Yaskawa INFORM job: pipe_uncentered_cylinder_program.JBI

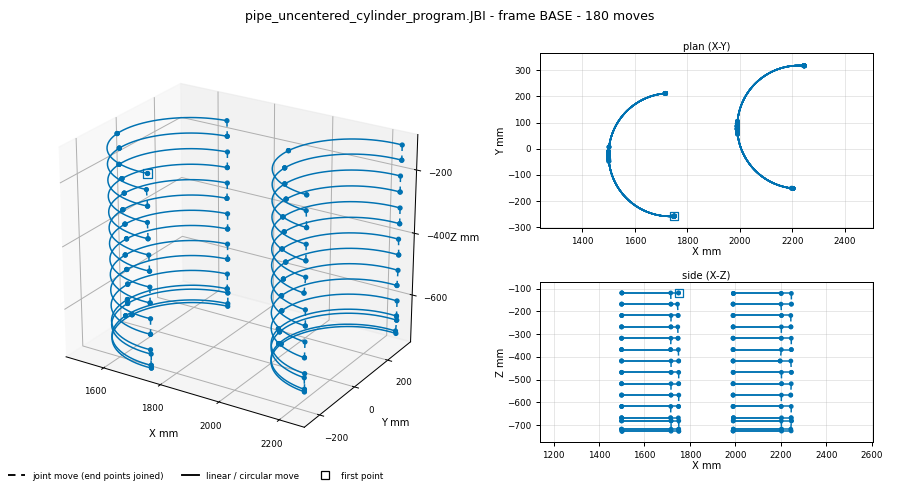
[picture p0: tool path of pipe_uncentered_cylinder_program.JBI in frame BASE, 180 of 245 moves have a stored position in this frame; points joined in program order, loops and branches not executed]
/JOB
//NAME pipe_uncentered_cylinder_program
//POS
///NPOS 240,0,240,0,0,0
///TOOL 0
///POSTYPE BASE
///RECTAN
///RCONF 0,0,0,0,0,0,0,0,0,0,0,0,0,0,0,0,0,0,0,0,0,0,0,0
C00000=1749.940904,-257.239351,-118.539050,-86.127714,-90.000000,5.000000
C00001=1749.940904,-257.239351,-118.539050,-86.127714,-90.000000,5.000000
C00002=1591.453481,-209.463262,-118.539050,-127.423189,-89.999999,5.000000
C00003=1500.680855,-47.796008,-118.539050,-173.950296,-90.000000,5.000000
C00004=1500.680855,-47.796008,-118.539050,-173.950296,-90.000000,5.000000
C00005=1500.680855,-47.796008,-118.539050,-173.950296,-90.000000,5.000000
C00006=1545.974830,117.313444,-118.539050,143.269507,-90.000000,5.000000
C00007=1715.536670,210.922784,-118.539050,94.533692,-90.000000,5.000000
C00008=1716.466846,210.994681,-167.787500,94.305952,-89.999999,5.000000
C00009=1716.466846,210.994681,-167.787500,94.305952,-89.999999,5.000000
C00010=1554.324971,127.859099,-167.787500,139.985523,-89.999999,5.000000
C00011=1499.816295,-37.466638,-167.787500,-175.000000,-90.000000,5.000000
C00012=1499.816295,-37.466638,-167.787500,-175.000000,-90.000000,5.000000
C00013=1499.816295,-37.466638,-167.787500,-175.000000,-90.000000,5.000000
C00014=1575.986813,-196.538427,-167.787500,-132.344944,-90.000000,5.000000
C00015=1745.242286,-257.510095,-167.787500,-87.276599,-90.000000,5.000000
C00016=1747.956735,-257.365215,-217.741000,-86.613037,-90.000000,5.000000
C00017=1747.956735,-257.365215,-217.741000,-86.613037,-90.000000,5.000000
C00018=1577.099305,-197.545821,-217.741000,-131.978582,-89.999999,5.000000
C00019=1500.085421,-41.323879,-217.741000,-175.000000,-89.999999,5.000000
C00020=1500.085421,-41.323879,-217.741000,-175.000000,-89.999999,5.000000
C00021=1500.085421,-41.323879,-217.741000,-175.000000,-89.999999,5.000000
C00022=1562.652474,137.256037,-217.741000,136.920187,-90.000000,5.000000
C00023=1717.040812,211.037190,-217.741000,94.165460,-90.000000,5.000000
C00024=1716.357109,210.986393,-267.822500,94.332816,-90.000000,5.000000
C00025=1716.357109,210.986393,-267.822500,94.332816,-90.000000,5.000000
C00026=1562.860730,137.478452,-267.822500,136.845809,-90.000000,5.000000
C00027=1499.417640,-27.601325,-267.822500,-175.000000,-90.000000,5.000000
C00028=1499.417640,-27.601325,-267.822500,-175.000000,-90.000000,5.000000
C00029=1499.417640,-27.601325,-267.822500,-175.000000,-90.000000,5.000000
C00030=1572.172718,-192.984054,-267.822500,-133.617628,-90.000000,5.000000
C00031=1746.492309,-257.447293,-267.822500,-86.971075,-90.000000,5.000000
C00032=1747.500808,-257.391753,-317.748500,-86.724521,-90.000000,5.000000
C00033=1747.500808,-257.391753,-317.748500,-86.724521,-90.000000,5.000000
C00034=1571.275066,-192.124158,-317.748500,-133.921067,-89.999999,5.000000
C00035=1499.445999,-17.233020,-317.748500,175.000000,-90.000000,5.000000
C00036=1499.445999,-17.233020,-317.748500,175.000000,-90.000000,5.000000
C00037=1499.445999,-17.233020,-317.748500,175.000000,-90.000000,5.000000
C00038=1566.953470,141.735162,-317.748500,135.404299,-90.000000,5.000000
C00039=1716.359373,210.986564,-317.748500,94.332262,-90.000000,5.000000
C00040=1715.055844,210.884161,-367.795500,94.651443,-90.000000,5.000000
C00041=1715.055844,210.884161,-367.795500,94.651443,-90.000000,5.000000
C00042=1568.265848,143.055676,-367.795500,134.949834,-89.999999,5.000000
C00043=1499.396571,-26.336761,-367.795500,-175.000000,-89.999999,5.000000
C00044=1499.396571,-26.336761,-367.795500,-175.000000,-89.999999,5.000000
C00045=1499.396571,-26.336761,-367.795500,-175.000000,-89.999999,5.000000
C00046=1569.975341,-190.862783,-367.795500,-134.363188,-90.000000,5.000000
C00047=1748.987493,-257.301936,-367.795500,-86.360949,-90.000000,5.000000
C00048=1750.526532,-257.198976,-417.775000,-85.984419,-90.000000,5.000000
C00049=1750.526532,-257.198976,-417.775000,-85.984419,-90.000000,5.000000
C00050=1569.600086,-190.494955,-417.775000,-134.491458,-90.000000,5.000000
C00051=1499.446271,-17.222088,-417.775000,175.000000,-90.000000,5.000000
C00052=1499.446271,-17.222088,-417.775000,175.000000,-90.000000,5.000000
C00053=1499.446271,-17.222088,-417.775000,175.000000,-90.000000,5.000000
C00054=1570.664090,145.415647,-417.775000,134.128488,-90.000000,5.000000
C00055=1716.962407,211.031467,-417.775000,94.184650,-90.000000,5.000000
C00056=1717.005411,211.034610,-467.823500,94.174124,-90.000000,5.000000
C00057=1717.005411,211.034610,-467.823500,94.174124,-90.000000,5.000000
C00058=1563.073398,137.704983,-467.823500,136.769961,-89.999999,5.000000
C00059=1499.674917,-11.171269,-467.823500,175.000000,-90.000000,5.000000
C00060=1499.674917,-11.171269,-467.823500,175.000000,-90.000000,5.000000
C00061=1499.674917,-11.171269,-467.823500,175.000000,-90.000000,5.000000
C00062=1571.299255,-192.147450,-467.823500,-133.912870,-90.000000,5.000000
C00063=1750.593496,-257.194266,-467.823500,-85.968032,-90.000000,5.000000
C00064=1750.562997,-257.196413,-517.742500,-85.975495,-90.000000,5.000000
C00065=1750.562997,-257.196413,-517.742500,-85.975495,-90.000000,5.000000
C00066=1569.533050,-190.429072,-517.742500,-134.514402,-90.000000,5.000000
C00067=1499.402780,-19.363326,-517.742500,175.000000,-89.999999,5.000000
C00068=1499.402780,-19.363326,-517.742500,175.000000,-89.999999,5.000000
C00069=1499.402780,-19.363326,-517.742500,175.000000,-89.999999,5.000000
C00070=1567.369334,142.155874,-517.742500,135.259896,-89.999999,5.000000
C00071=1716.613272,211.005660,-517.742500,94.270109,-89.999999,5.000000
C00072=1716.823581,211.021268,-567.815000,94.218629,-90.000000,5.000000
C00073=1716.823581,211.021268,-567.815000,94.218629,-90.000000,5.000000
C00074=1567.685117,142.473927,-567.815000,135.150489,-90.000000,5.000000
C00075=1499.562947,-13.635054,-567.815000,175.000000,-89.999999,5.000000
C00076=1499.562947,-13.635054,-567.815000,175.000000,-89.999999,5.000000
C00077=1499.562947,-13.635054,-567.815000,175.000000,-89.999999,5.000000
C00078=1560.121142,-180.623494,-567.815000,-137.832681,-90.000000,5.000000
C00079=1751.024331,-257.163499,-567.815000,-85.862594,-90.000000,5.000000
C00080=1750.015796,-257.234270,-617.780500,-86.109390,-89.999999,5.000000
C00081=1750.015796,-257.234270,-617.780500,-86.109390,-89.999999,5.000000
C00082=1559.512787,-179.949185,-617.780500,-138.054373,-90.000000,5.000000
C00083=1499.705471,-10.583354,-617.780500,175.000000,-90.000000,5.000000
C00084=1499.705471,-10.583354,-617.780500,175.000000,-90.000000,5.000000
C00085=1499.705471,-10.583354,-617.780500,175.000000,-90.000000,5.000000
C00086=1570.812903,145.559872,-617.780500,134.077900,-90.000000,5.000000
C00087=1715.782793,210.942170,-617.780500,94.473426,-89.999999,5.000000
C00088=1715.115153,210.888979,-667.838500,94.636917,-90.000000,5.000000
C00089=1715.115153,210.888979,-667.838500,94.636917,-90.000000,5.000000
C00090=1572.298871,146.986185,-667.838500,133.575106,-90.000000,5.000000
C00091=1499.565682,-13.567229,-667.838500,175.000000,-90.000000,5.000000
C00092=1499.565682,-13.567229,-667.838500,175.000000,-90.000000,5.000000
C00093=1499.565682,-13.567229,-667.838500,175.000000,-90.000000,5.000000
C00094=1567.110596,-188.012358,-667.838500,-135.349696,-90.000000,5.000000
C00095=1749.049055,-257.298013,-667.838500,-86.345891,-90.000000,5.000000
C00096=1750.503472,-257.200594,-717.761000,-85.990062,-90.000000,5.000000
C00097=1750.503472,-257.200594,-717.761000,-85.990062,-90.000000,5.000000
C00098=1567.704779,-188.611679,-717.761000,-135.143684,-90.000000,5.000000
C00099=1499.381472,-24.971037,-717.761000,-175.000000,-90.000000,5.000000
C00100=1499.381472,-24.971037,-717.761000,-175.000000,-90.000000,5.000000
C00101=1499.381472,-24.971037,-717.761000,-175.000000,-90.000000,5.000000
C00102=1562.233334,136.806640,-717.761000,137.070196,-90.000000,5.000000
C00103=1717.054447,211.038183,-717.761000,94.162123,-89.999999,5.000000
C00104=1717.121726,211.043069,-681.141960,-175.000000,-60.000000,-85.854344
C00105=1717.121726,211.043069,-681.141960,-175.000000,-60.000000,-85.854344
C00106=1567.606056,142.394412,-681.141960,-175.000000,-60.000000,-44.822139
C00107=1499.579001,-13.243673,-681.141960,175.000000,-60.000000,-5.000000
C00108=1499.579001,-13.243673,-681.141960,175.000000,-60.000000,-5.000000
C00109=1499.579001,-13.243673,-681.141960,175.000000,-60.000000,-5.000000
C00110=1566.014614,-186.895493,-681.141960,175.000000,-60.000000,44.268328
C00111=1750.849014,-257.176115,-681.141960,175.000000,-60.000000,94.094499
C00112=1751.015595,-257.164131,-726.640960,175.000000,-60.000000,94.135268
C00113=1751.015595,-257.164131,-726.640960,175.000000,-60.000000,94.135268
C00114=1552.700260,-172.020396,-726.640960,-175.000000,-60.000000,39.393640
C00115=1501.257028,6.615173,-726.640960,175.000000,-60.000000,-7.263097
C00116=1501.257028,6.615173,-726.640960,175.000000,-60.000000,-7.263097
C00117=1501.257028,6.615173,-726.640960,175.000000,-60.000000,-7.263097
C00118=1579.136007,153.239023,-726.640960,175.000000,-60.000000,-48.686744
C00119=1716.838691,211.022382,-726.640960,-175.000000,-60.000000,-85.785069
C00120=2201.495182,-151.068736,-120.674700,-95.658348,-90.000000,5.000000
C00121=2201.495182,-151.068736,-120.674700,-95.658348,-90.000000,5.000000
C00122=2044.257197,-67.678403,-120.674700,-140.219665,-90.000000,5.000000
C00123=1990.979209,104.765230,-120.674700,174.557660,-90.000000,5.000000
C00124=1990.979209,104.765230,-120.674700,174.557660,-90.000000,5.000000
C00125=1990.979209,104.765230,-120.674700,174.557660,-90.000000,5.000000
C00126=2064.299554,253.919936,-120.674700,133.087419,-90.000000,5.000000
C00127=2246.112616,316.235511,-120.674700,84.750402,-90.000000,5.000000
C00128=2246.169004,316.230323,-167.736500,84.736579,-90.000000,5.000000
C00129=2246.169004,316.230323,-167.736500,84.736579,-90.000000,5.000000
C00130=2063.146664,252.834241,-167.736500,133.473995,-90.000000,5.000000
C00131=1989.947901,86.047865,-167.736500,175.000000,-89.999999,5.000000
C00132=1989.947901,86.047865,-167.736500,175.000000,-89.999999,5.000000
C00133=1989.947901,86.047865,-167.736500,175.000000,-89.999999,5.000000
C00134=2052.059148,-76.582521,-167.736500,-137.329465,-89.999999,5.000000
C00135=2200.564996,-150.974703,-167.736500,-95.886570,-90.000000,5.000000
C00136=2202.695265,-151.184528,-217.738500,-95.364039,-89.999999,5.000000
C00137=2202.695265,-151.184528,-217.738500,-95.364039,-89.999999,5.000000
C00138=2049.346534,-73.588554,-217.738500,-138.315683,-90.000000,5.000000
C00139=1989.967085,87.147586,-217.738500,175.000000,-90.000000,5.000000
C00140=1989.967085,87.147586,-217.738500,175.000000,-90.000000,5.000000
C00141=1989.967085,87.147586,-217.738500,175.000000,-90.000000,5.000000
C00142=2060.819888,250.597642,-217.738500,134.261837,-89.999999,5.000000
C00143=2243.608192,316.452099,-217.738500,85.364033,-90.000000,5.000000
C00144=2244.039674,316.416710,-267.790000,85.258352,-90.000000,5.000000
C00145=2244.039674,316.416710,-267.790000,85.258352,-90.000000,5.000000
C00146=2071.779846,260.622536,-267.790000,130.635454,-89.999999,5.000000
C00147=1990.257189,95.059201,-267.790000,175.000000,-89.999999,5.000000
C00148=1990.257189,95.059201,-267.790000,175.000000,-89.999999,5.000000
C00149=1990.257189,95.059201,-267.790000,175.000000,-89.999999,5.000000
C00150=2049.513988,-73.776402,-267.790000,-138.254254,-90.000000,5.000000
C00151=2202.070096,-151.124984,-267.790000,-95.517338,-89.999999,5.000000
C00152=2201.732367,-151.092115,-317.761500,-95.600169,-90.000000,5.000000
C00153=2201.732367,-151.092115,-317.761500,-95.600169,-90.000000,5.000000
C00154=2058.339900,-83.136929,-317.761500,-135.113353,-90.000000,5.000000
C00155=1989.951054,78.756762,-317.761500,-175.000000,-90.000000,5.000000
C00156=1989.951054,78.756762,-317.761500,-175.000000,-90.000000,5.000000
C00157=1989.951054,78.756762,-317.761500,-175.000000,-90.000000,5.000000
C00158=2070.732503,259.718356,-317.761500,130.973211,-90.000000,5.000000
C00159=2245.637578,316.278670,-317.761500,84.866839,-90.000000,5.000000
C00160=2246.012474,316.244690,-367.767000,84.774950,-89.999999,5.000000
C00161=2246.012474,316.244690,-367.767000,84.774950,-89.999999,5.000000
C00162=2061.479430,251.237892,-367.767000,134.037456,-89.999999,5.000000
C00163=1989.955586,86.524700,-367.767000,175.000000,-90.000000,5.000000
C00164=1989.955586,86.524700,-367.767000,175.000000,-90.000000,5.000000
C00165=1989.955586,86.524700,-367.767000,175.000000,-90.000000,5.000000
C00166=2045.484077,-69.139856,-367.767000,-139.753869,-89.999999,5.000000
C00167=2201.922845,-151.110713,-367.767000,-95.553451,-90.000000,5.000000
C00168=2196.726495,-150.546997,-417.788500,-96.829383,-90.000000,5.000000
C00169=2196.726495,-150.546997,-417.788500,-96.829383,-90.000000,5.000000
C00170=2053.431275,-78.058253,-417.788500,-136.837571,-90.000000,5.000000
C00171=1990.036838,75.135124,-417.788500,-175.000000,-89.999999,5.000000
C00172=1990.036838,75.135124,-417.788500,-175.000000,-89.999999,5.000000
C00173=1990.036838,75.135124,-417.788500,-175.000000,-89.999999,5.000000
C00174=2058.402661,248.207538,-417.788500,135.091648,-90.000000,5.000000
C00175=2243.881899,316.429743,-417.788500,85.296997,-89.999999,5.000000
C00176=2246.061371,316.240213,-467.763000,84.762964,-90.000000,5.000000
C00177=2246.061371,316.240213,-467.763000,84.762964,-90.000000,5.000000
C00178=2071.679385,260.536273,-467.763000,130.667777,-90.000000,5.000000
C00179=1990.326877,96.298740,-467.763000,175.000000,-90.000000,5.000000
C00180=1990.326877,96.298740,-467.763000,175.000000,-90.000000,5.000000
C00181=1990.326877,96.298740,-467.763000,175.000000,-90.000000,5.000000
C00182=2052.360794,-76.909127,-467.763000,-137.220937,-90.000000,5.000000
C00183=2202.313125,-151.148331,-467.763000,-95.457740,-90.000000,5.000000
C00184=2202.902488,-151.203892,-517.762500,-95.313234,-90.000000,5.000000
C00185=2202.902488,-151.203892,-517.762500,-95.313234,-90.000000,5.000000
C00186=2057.105877,-81.888713,-517.762500,-135.541819,-89.999999,5.000000
C00187=1989.931219,84.678581,-517.762500,175.000000,-89.999999,5.000000
C00188=1989.931219,84.678581,-517.762500,175.000000,-89.999999,5.000000
C00189=1989.931219,84.678581,-517.762500,175.000000,-89.999999,5.000000
C00190=2068.385658,257.652621,-517.762500,131.736413,-89.999999,5.000000
C00191=2245.482409,316.292557,-517.762500,84.904869,-90.000000,5.000000
C00192=2243.362690,316.471877,-567.772500,85.424156,-90.000000,5.000000
C00193=2243.362690,316.471877,-567.772500,85.424156,-90.000000,5.000000
C00194=2051.378042,240.848086,-567.772500,137.575342,-90.000000,5.000000
C00195=1990.060890,74.405537,-567.772500,-175.000000,-89.999999,5.000000
C00196=1990.060890,74.405537,-567.772500,-175.000000,-89.999999,5.000000
C00197=1990.060890,74.405537,-567.772500,-175.000000,-89.999999,5.000000
C00198=2061.322668,-86.078546,-567.772500,-134.090710,-89.999999,5.000000
C00199=2202.327386,-151.149694,-567.772500,-95.454242,-90.000000,5.000000
C00200=2201.367177,-151.056018,-617.754500,-95.689749,-90.000000,5.000000
C00201=2201.367177,-151.056018,-617.754500,-95.689749,-90.000000,5.000000
C00202=2052.658725,-77.230498,-617.754500,-137.113963,-90.000000,5.000000
C00203=1989.999951,76.421959,-617.754500,-175.000000,-89.999999,5.000000
C00204=1989.999951,76.421959,-617.754500,-175.000000,-89.999999,5.000000
C00205=1989.999951,76.421959,-617.754500,-175.000000,-89.999999,5.000000
C00206=2056.480347,246.256427,-617.754500,135.760260,-90.000000,5.000000
C00207=2245.513226,316.289808,-617.754500,84.897316,-90.000000,5.000000
C00208=2245.267041,316.311660,-667.687000,84.957648,-90.000000,5.000000
C00209=2245.267041,316.311660,-667.687000,84.957648,-90.000000,5.000000
C00210=2046.291839,235.096654,-667.687000,139.449624,-90.000000,5.000000
C00211=1991.451727,55.742592,-667.687000,-173.453172,-89.999999,5.000000
C00212=1991.451727,55.742592,-667.687000,-173.453172,-89.999999,5.000000
C00213=1991.451727,55.742592,-667.687000,-173.453172,-89.999999,5.000000
C00214=2061.762417,-86.503446,-667.687000,-133.941441,-90.000000,5.000000
C00215=2202.791447,-151.193539,-667.687000,-95.340457,-90.000000,5.000000
C00216=2202.766975,-151.191250,-717.769500,-95.346457,-89.999999,5.000000
C00217=2202.766975,-151.191250,-717.769500,-95.346457,-89.999999,5.000000
C00218=2056.491256,-81.260006,-717.769500,-135.756443,-90.000000,5.000000
C00219=1991.056336,59.447196,-717.769500,-174.362636,-89.999999,5.000000
C00220=1991.056336,59.447196,-717.769500,-174.362636,-89.999999,5.000000
C00221=1991.056336,59.447196,-717.769500,-174.362636,-89.999999,5.000000
C00222=2050.583896,239.974736,-717.769500,137.863492,-90.000000,5.000000
C00223=2243.561805,316.455856,-717.769500,85.375394,-89.999999,5.000000
C00224=2246.301849,316.218047,-681.093960,175.000000,-60.000000,-95.295987
C00225=2246.301849,316.218047,-681.093960,175.000000,-60.000000,-95.295987
C00226=2049.280658,238.522168,-681.093960,-175.000000,-60.000000,-41.660131
C00227=1990.652766,63.985921,-681.093960,175.000000,-60.000000,5.000000
C00228=1990.652766,63.985921,-681.093960,175.000000,-60.000000,5.000000
C00229=1990.652766,63.985921,-681.093960,175.000000,-60.000000,5.000000
C00230=2060.887500,-85.655884,-681.093960,175.000000,-60.000000,45.761205
C00231=2201.648298,-151.083856,-681.093960,175.000000,-60.000000,84.379210
C00232=2202.847007,-151.198726,-725.482960,-175.000000,-60.000000,84.673164
C00233=2202.847007,-151.198726,-725.482960,-175.000000,-60.000000,84.673164
C00234=2065.711002,-90.221730,-725.482960,-175.000000,-60.000000,47.382559
C00235=1990.062143,74.369326,-725.482960,175.000000,-60.000000,5.000000
C00236=1990.062143,74.369326,-725.482960,175.000000,-60.000000,5.000000
C00237=1990.062143,74.369326,-725.482960,175.000000,-60.000000,5.000000
C00238=2051.419035,240.892928,-725.482960,175.000000,-60.000000,-42.439489
C00239=2245.154859,316.321531,-725.482960,175.000000,-60.000000,-95.014862
///POSTYPE PULSE
///PULSE
EX00000=80896.0
EX00001=256000.0
///POSTYPE PULSE
///PULSE
EC00000=80896.0
EC00001=80896.0
EC00002=80896.0
EC00003=80896.0
EC00004=80896.0
EC00005=80896.0
EC00006=80896.0
EC00007=80896.0
EC00008=80896.0
EC00009=80896.0
EC00010=80896.0
EC00011=80896.0
EC00012=80896.0
EC00013=80896.0
EC00014=80896.0
EC00015=80896.0
EC00016=80896.0
EC00017=80896.0
EC00018=80896.0
EC00019=80896.0
EC00020=80896.0
EC00021=80896.0
EC00022=80896.0
EC00023=80896.0
EC00024=80896.0
EC00025=80896.0
EC00026=80896.0
EC00027=80896.0
EC00028=80896.0
EC00029=80896.0
EC00030=80896.0
EC00031=80896.0
EC00032=80896.0
EC00033=80896.0
EC00034=80896.0
EC00035=80896.0
EC00036=80896.0
EC00037=80896.0
EC00038=80896.0
EC00039=80896.0
EC00040=80896.0
EC00041=80896.0
EC00042=80896.0
EC00043=80896.0
EC00044=80896.0
EC00045=80896.0
EC00046=80896.0
EC00047=80896.0
EC00048=80896.0
EC00049=80896.0
EC00050=80896.0
EC00051=80896.0
EC00052=80896.0
EC00053=80896.0
EC00054=80896.0
EC00055=80896.0
EC00056=80896.0
EC00057=80896.0
EC00058=80896.0
EC00059=80896.0
EC00060=80896.0
EC00061=80896.0
EC00062=80896.0
EC00063=80896.0
EC00064=80896.0
EC00065=80896.0
EC00066=80896.0
EC00067=80896.0
EC00068=80896.0
EC00069=80896.0
EC00070=80896.0
EC00071=80896.0
EC00072=80896.0
EC00073=80896.0
EC00074=80896.0
EC00075=80896.0
EC00076=80896.0
EC00077=80896.0
EC00078=80896.0
EC00079=80896.0
EC00080=80896.0
EC00081=80896.0
EC00082=80896.0
EC00083=80896.0
EC00084=80896.0
EC00085=80896.0
EC00086=80896.0
EC00087=80896.0
EC00088=80896.0
EC00089=80896.0
EC00090=80896.0
EC00091=80896.0
EC00092=80896.0
EC00093=80896.0
EC00094=80896.0
EC00095=80896.0
EC00096=80896.0
EC00097=80896.0
EC00098=80896.0
EC00099=80896.0
EC00100=80896.0
EC00101=80896.0
EC00102=80896.0
EC00103=80896.0
EC00104=80896.0
EC00105=80896.0
EC00106=80896.0
EC00107=80896.0
EC00108=80896.0
EC00109=80896.0
EC00110=80896.0
EC00111=80896.0
EC00112=80896.0
EC00113=80896.0
EC00114=80896.0
EC00115=80896.0
EC00116=80896.0
EC00117=80896.0
EC00118=80896.0
EC00119=80896.0
EC00120=256000.0
EC00121=256000.0
EC00122=256000.0
EC00123=256000.0
EC00124=256000.0
EC00125=256000.0
EC00126=256000.0
EC00127=256000.0
EC00128=256000.0
EC00129=256000.0
EC00130=256000.0
EC00131=256000.0
EC00132=256000.0
EC00133=256000.0
EC00134=256000.0
EC00135=256000.0
EC00136=256000.0
EC00137=256000.0
EC00138=256000.0
EC00139=256000.0
EC00140=256000.0
EC00141=256000.0
EC00142=256000.0
EC00143=256000.0
EC00144=256000.0
EC00145=256000.0
EC00146=256000.0
EC00147=256000.0
EC00148=256000.0
EC00149=256000.0
EC00150=256000.0
EC00151=256000.0
EC00152=256000.0
EC00153=256000.0
EC00154=256000.0
EC00155=256000.0
EC00156=256000.0
EC00157=256000.0
EC00158=256000.0
EC00159=256000.0
EC00160=256000.0
EC00161=256000.0
EC00162=256000.0
EC00163=256000.0
EC00164=256000.0
EC00165=256000.0
EC00166=256000.0
EC00167=256000.0
EC00168=256000.0
EC00169=256000.0
EC00170=256000.0
EC00171=256000.0
EC00172=256000.0
EC00173=256000.0
EC00174=256000.0
EC00175=256000.0
EC00176=256000.0
EC00177=256000.0
EC00178=256000.0
EC00179=256000.0
EC00180=256000.0
EC00181=256000.0
EC00182=256000.0
EC00183=256000.0
EC00184=256000.0
EC00185=256000.0
EC00186=256000.0
EC00187=256000.0
EC00188=256000.0
EC00189=256000.0
EC00190=256000.0
EC00191=256000.0
EC00192=256000.0
EC00193=256000.0
EC00194=256000.0
EC00195=256000.0
EC00196=256000.0
EC00197=256000.0
EC00198=256000.0
EC00199=256000.0
EC00200=256000.0
EC00201=256000.0
EC00202=256000.0
EC00203=256000.0
EC00204=256000.0
EC00205=256000.0
EC00206=256000.0
EC00207=256000.0
EC00208=256000.0
EC00209=256000.0
EC00210=256000.0
EC00211=256000.0
EC00212=256000.0
EC00213=256000.0
EC00214=256000.0
EC00215=256000.0
EC00216=256000.0
EC00217=256000.0
EC00218=256000.0
EC00219=256000.0
EC00220=256000.0
EC00221=256000.0
EC00222=256000.0
EC00223=256000.0
EC00224=256000.0
EC00225=256000.0
EC00226=256000.0
EC00227=256000.0
EC00228=256000.0
EC00229=256000.0
EC00230=256000.0
EC00231=256000.0
EC00232=256000.0
EC00233=256000.0
EC00234=256000.0
EC00235=256000.0
EC00236=256000.0
EC00237=256000.0
EC00238=256000.0
EC00239=256000.0
//INST
///DATE 2023/08/15 14:21
///ATTR SC,RW,RJ
////FRAME BASE
///GROUP1 RB1,ST1
NOP
MOVJ P009 EX000 VJ=15.00
MOVJ C00000 EC00000 VJ=15.0
CALL JOB:SPYON
MOVC C00001 EC00001 V=150.0
MOVC C00002 EC00002 V=150.0
MOVC C00003 EC00003 V=150.0
MOVJ C00004 EC00004 VJ=15.0
MOVC C00005 EC00005 V=150.0
MOVC C00006 EC00006 V=150.0
MOVC C00007 EC00007 V=150.0
MOVJ C00008 EC00008 VJ=15.0
MOVC C00009 EC00009 V=150.0
MOVC C00010 EC00010 V=150.0
MOVC C00011 EC00011 V=150.0
MOVJ C00012 EC00012 VJ=15.0
MOVC C00013 EC00013 V=150.0
MOVC C00014 EC00014 V=150.0
MOVC C00015 EC00015 V=150.0
MOVJ C00016 EC00016 VJ=15.0
MOVC C00017 EC00017 V=150.0
MOVC C00018 EC00018 V=150.0
MOVC C00019 EC00019 V=150.0
MOVJ C00020 EC00020 VJ=15.0
MOVC C00021 EC00021 V=150.0
MOVC C00022 EC00022 V=150.0
MOVC C00023 EC00023 V=150.0
MOVJ C00024 EC00024 VJ=15.0
MOVC C00025 EC00025 V=150.0
MOVC C00026 EC00026 V=150.0
MOVC C00027 EC00027 V=150.0
MOVJ C00028 EC00028 VJ=15.0
MOVC C00029 EC00029 V=150.0
MOVC C00030 EC00030 V=150.0
MOVC C00031 EC00031 V=150.0
MOVJ C00032 EC00032 VJ=15.0
MOVC C00033 EC00033 V=150.0
MOVC C00034 EC00034 V=150.0
MOVC C00035 EC00035 V=150.0
MOVJ C00036 EC00036 VJ=15.0
MOVC C00037 EC00037 V=150.0
MOVC C00038 EC00038 V=150.0
MOVC C00039 EC00039 V=150.0
MOVJ C00040 EC00040 VJ=15.0
MOVC C00041 EC00041 V=150.0
MOVC C00042 EC00042 V=150.0
MOVC C00043 EC00043 V=150.0
MOVJ C00044 EC00044 VJ=15.0
MOVC C00045 EC00045 V=150.0
MOVC C00046 EC00046 V=150.0
MOVC C00047 EC00047 V=150.0
MOVJ C00048 EC00048 VJ=15.0
MOVC C00049 EC00049 V=150.0
MOVC C00050 EC00050 V=150.0
MOVC C00051 EC00051 V=150.0
MOVJ C00052 EC00052 VJ=15.0
MOVC C00053 EC00053 V=150.0
MOVC C00054 EC00054 V=150.0
MOVC C00055 EC00055 V=150.0
MOVJ C00056 EC00056 VJ=15.0
MOVC C00057 EC00057 V=150.0
MOVC C00058 EC00058 V=150.0
MOVC C00059 EC00059 V=150.0
MOVJ C00060 EC00060 VJ=15.0
MOVC C00061 EC00061 V=150.0
MOVC C00062 EC00062 V=150.0
MOVC C00063 EC00063 V=150.0
MOVJ C00064 EC00064 VJ=15.0
MOVC C00065 EC00065 V=150.0
MOVC C00066 EC00066 V=150.0
MOVC C00067 EC00067 V=150.0
MOVJ C00068 EC00068 VJ=15.0
MOVC C00069 EC00069 V=150.0
MOVC C00070 EC00070 V=150.0
MOVC C00071 EC00071 V=150.0
MOVJ C00072 EC00072 VJ=15.0
MOVC C00073 EC00073 V=150.0
MOVC C00074 EC00074 V=150.0
MOVC C00075 EC00075 V=150.0
MOVJ C00076 EC00076 VJ=15.0
MOVC C00077 EC00077 V=150.0
MOVC C00078 EC00078 V=150.0
MOVC C00079 EC00079 V=150.0
MOVJ C00080 EC00080 VJ=15.0
MOVC C00081 EC00081 V=150.0
MOVC C00082 EC00082 V=150.0
MOVC C00083 EC00083 V=150.0
MOVJ C00084 EC00084 VJ=15.0
MOVC C00085 EC00085 V=150.0
MOVC C00086 EC00086 V=150.0
MOVC C00087 EC00087 V=150.0
MOVJ C00088 EC00088 VJ=15.0
MOVC C00089 EC00089 V=150.0
MOVC C00090 EC00090 V=150.0
MOVC C00091 EC00091 V=150.0
MOVJ C00092 EC00092 VJ=15.0
MOVC C00093 EC00093 V=150.0
MOVC C00094 EC00094 V=150.0
MOVC C00095 EC00095 V=150.0
MOVJ C00096 EC00096 VJ=15.0
MOVC C00097 EC00097 V=150.0
MOVC C00098 EC00098 V=150.0
MOVC C00099 EC00099 V=150.0
MOVJ C00100 EC00100 VJ=15.0
MOVC C00101 EC00101 V=150.0
MOVC C00102 EC00102 V=150.0
MOVC C00103 EC00103 V=150.0
MOVJ C00104 EC00104 VJ=15.0
MOVC C00105 EC00105 V=150.0
MOVC C00106 EC00106 V=150.0
MOVC C00107 EC00107 V=150.0
MOVJ C00108 EC00108 VJ=15.0
MOVC C00109 EC00109 V=150.0
MOVC C00110 EC00110 V=150.0
MOVC C00111 EC00111 V=150.0
MOVJ C00112 EC00112 VJ=15.0
MOVC C00113 EC00113 V=150.0
MOVC C00114 EC00114 V=150.0
MOVC C00115 EC00115 V=150.0
MOVJ C00116 EC00116 VJ=15.0
MOVC C00117 EC00117 V=150.0
MOVC C00118 EC00118 V=150.0
MOVC C00119 EC00119 V=150.0
CALL JOB:SPYOF
MOVJ P009 VJ=15.00
MOVL P009 EX00000 V=150.0
MOVJ C00120 EC00120 VJ=15.0
CALL JOB:SPYON
MOVC C00121 EC00121 V=150.0
MOVC C00122 EC00122 V=150.0
MOVC C00123 EC00123 V=150.0
MOVJ C00124 EC00124 VJ=15.0
MOVC C00125 EC00125 V=150.0
MOVC C00126 EC00126 V=150.0
MOVC C00127 EC00127 V=150.0
MOVJ C00128 EC00128 VJ=15.0
MOVC C00129 EC00129 V=150.0
MOVC C00130 EC00130 V=150.0
MOVC C00131 EC00131 V=150.0
MOVJ C00132 EC00132 VJ=15.0
MOVC C00133 EC00133 V=150.0
MOVC C00134 EC00134 V=150.0
MOVC C00135 EC00135 V=150.0
MOVJ C00136 EC00136 VJ=15.0
MOVC C00137 EC00137 V=150.0
MOVC C00138 EC00138 V=150.0
MOVC C00139 EC00139 V=150.0
MOVJ C00140 EC00140 VJ=15.0
MOVC C00141 EC00141 V=150.0
MOVC C00142 EC00142 V=150.0
MOVC C00143 EC00143 V=150.0
MOVJ C00144 EC00144 VJ=15.0
MOVC C00145 EC00145 V=150.0
MOVC C00146 EC00146 V=150.0
MOVC C00147 EC00147 V=150.0
MOVJ C00148 EC00148 VJ=15.0
MOVC C00149 EC00149 V=150.0
MOVC C00150 EC00150 V=150.0
MOVC C00151 EC00151 V=150.0
MOVJ C00152 EC00152 VJ=15.0
MOVC C00153 EC00153 V=150.0
MOVC C00154 EC00154 V=150.0
MOVC C00155 EC00155 V=150.0
MOVJ C00156 EC00156 VJ=15.0
MOVC C00157 EC00157 V=150.0
MOVC C00158 EC00158 V=150.0
MOVC C00159 EC00159 V=150.0
MOVJ C00160 EC00160 VJ=15.0
MOVC C00161 EC00161 V=150.0
MOVC C00162 EC00162 V=150.0
MOVC C00163 EC00163 V=150.0
MOVJ C00164 EC00164 VJ=15.0
MOVC C00165 EC00165 V=150.0
MOVC C00166 EC00166 V=150.0
MOVC C00167 EC00167 V=150.0
MOVJ C00168 EC00168 VJ=15.0
MOVC C00169 EC00169 V=150.0
MOVC C00170 EC00170 V=150.0
MOVC C00171 EC00171 V=150.0
MOVJ C00172 EC00172 VJ=15.0
MOVC C00173 EC00173 V=150.0
MOVC C00174 EC00174 V=150.0
MOVC C00175 EC00175 V=150.0
MOVJ C00176 EC00176 VJ=15.0
MOVC C00177 EC00177 V=150.0
MOVC C00178 EC00178 V=150.0
MOVC C00179 EC00179 V=150.0
MOVJ C00180 EC00180 VJ=15.0
MOVC C00181 EC00181 V=150.0
MOVC C00182 EC00182 V=150.0
MOVC C00183 EC00183 V=150.0
MOVJ C00184 EC00184 VJ=15.0
MOVC C00185 EC00185 V=150.0
MOVC C00186 EC00186 V=150.0
MOVC C00187 EC00187 V=150.0
MOVJ C00188 EC00188 VJ=15.0
MOVC C00189 EC00189 V=150.0
MOVC C00190 EC00190 V=150.0
MOVC C00191 EC00191 V=150.0
MOVJ C00192 EC00192 VJ=15.0
MOVC C00193 EC00193 V=150.0
MOVC C00194 EC00194 V=150.0
MOVC C00195 EC00195 V=150.0
MOVJ C00196 EC00196 VJ=15.0
MOVC C00197 EC00197 V=150.0
MOVC C00198 EC00198 V=150.0
MOVC C00199 EC00199 V=150.0
MOVJ C00200 EC00200 VJ=15.0
MOVC C00201 EC00201 V=150.0
MOVC C00202 EC00202 V=150.0
MOVC C00203 EC00203 V=150.0
MOVJ C00204 EC00204 VJ=15.0
MOVC C00205 EC00205 V=150.0
MOVC C00206 EC00206 V=150.0
MOVC C00207 EC00207 V=150.0
MOVJ C00208 EC00208 VJ=15.0
MOVC C00209 EC00209 V=150.0
MOVC C00210 EC00210 V=150.0
MOVC C00211 EC00211 V=150.0
MOVJ C00212 EC00212 VJ=15.0
MOVC C00213 EC00213 V=150.0
MOVC C00214 EC00214 V=150.0
MOVC C00215 EC00215 V=150.0
MOVJ C00216 EC00216 VJ=15.0
MOVC C00217 EC00217 V=150.0
MOVC C00218 EC00218 V=150.0
MOVC C00219 EC00219 V=150.0
MOVJ C00220 EC00220 VJ=15.0
MOVC C00221 EC00221 V=150.0
MOVC C00222 EC00222 V=150.0
MOVC C00223 EC00223 V=150.0
MOVJ C00224 EC00224 VJ=15.0
MOVC C00225 EC00225 V=150.0
MOVC C00226 EC00226 V=150.0
MOVC C00227 EC00227 V=150.0
MOVJ C00228 EC00228 VJ=15.0
MOVC C00229 EC00229 V=150.0
MOVC C00230 EC00230 V=150.0
MOVC C00231 EC00231 V=150.0
MOVJ C00232 EC00232 VJ=15.0
MOVC C00233 EC00233 V=150.0
MOVC C00234 EC00234 V=150.0
MOVC C00235 EC00235 V=150.0
MOVJ C00236 EC00236 VJ=15.0
MOVC C00237 EC00237 V=150.0
MOVC C00238 EC00238 V=150.0
MOVC C00239 EC00239 V=150.0
CALL JOB:SPYOF
MOVJ P009 VJ=15.00
MOVL P009 EX00001 V=150.0
END
